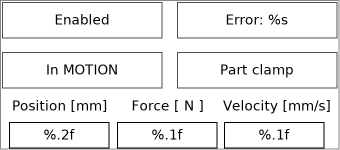
VISUALIZATION vHP3_AxisMainParams  // 340x150
VAR_IN_OUT
	fbAxis	: fbHP_Axis;
END_VAR
    Rectangle (9,122 100x26), "%.2f", text variable: fbAxis.McReadActualPosition.Position
    Label (10,93 100x26), "Position [mm]"
    Rectangle (117,122 100x26), "%.1f", text variable: fbAxis.fbForceFilter.rOut
    Label (118,93 100x26), "Force [ N ]"
    Rectangle (224,122 100x26), "%.1f", text variable: fbAxis.McReadActualVelocity.ActualVelocity, colour toggle: fbAxis.IsMoving
    Label (225,93 104x26), "Velocity [mm/s]"
    Rectangle (177,2 160x36), "Error: %s", text variable: TO_STRING(fbAxis.nActEvent), colour toggle: fbAxis.IsErrorActive
    Rectangle (2,2 160x36), "Enabled", colour toggle: fbAxis.Enabled
    Rectangle (2,52 160x36), "In MOTION", text variable: TO_STRING(fbAxis.nActEvent), colour toggle: fbAxis.IsMoving
    Rectangle (177,52 160x36), "Part clamp", text variable: TO_STRING(fbAxis.nActEvent), colour toggle: fbAxis.PartClamp
END_VISUALIZATION

(* stored: Version 1.1.0.1, ProductVersion 3.1.4024.12
   Visu vHP3_AxisMainParams: Id {c1c82617-8a94-4b3c-9acd-9b98687fb0b1} *)
